FUNCTION_BLOCK LC_TOUCH (* Composite Function Block Type *)
  (* Standard: 61499-2 *)
  (* Version 0.0, 2012-01-30, 4DIAC-IDE, 4DIAC-Consortium *)
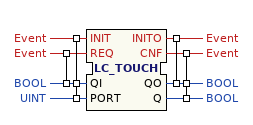
  EVENT_INPUT
    INIT WITH QI, PORT; (* Initialization Request *)
    REQ WITH QI; (* Normal Execution Request *)
  END_EVENT
  EVENT_OUTPUT
    INITO WITH QO; (* Initialization Confirm *)
    CNF WITH QO, Q; (* Execution Confirmation *)
  END_EVENT
  VAR_INPUT
    QI : BOOL; (* Input event qualifier *)
    PORT : UINT; (* Port # *)
  END_VAR
  VAR_OUTPUT
    QO : BOOL; (* Output event qualifier *)
    Q : BOOL; (* True if pressed *)
  END_VAR
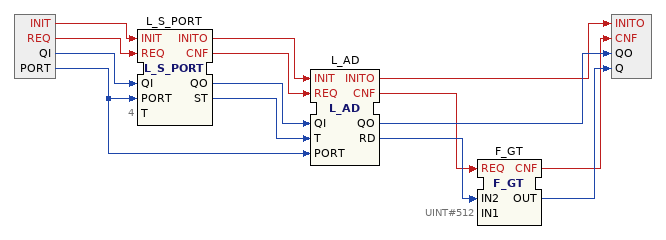
  FBS
    L_AD : L_AD;
    L_S_PORT : L_S_PORT(T := 4);
    F_GT : F_GT(IN1 := UINT#512);
  END_FBS
  EVENT_CONNECTIONS
    INIT TO L_S_PORT.INIT;
    L_S_PORT.INITO TO L_AD.INIT;
    L_AD.INITO TO INITO;
    REQ TO L_S_PORT.REQ;
    L_S_PORT.CNF TO L_AD.REQ;
    L_AD.CNF TO F_GT.REQ;
    F_GT.CNF TO CNF;
  END_CONNECTIONS
  DATA_CONNECTIONS
    L_AD.QO TO QO;
    L_S_PORT.QO TO L_AD.QI;
    L_S_PORT.ST TO L_AD.T;
    QI TO L_S_PORT.QI;
    PORT TO L_S_PORT.PORT;
    PORT TO L_AD.PORT;
    L_AD.RD TO F_GT.IN2;
    F_GT.OUT TO Q;
  END_CONNECTIONS
END_FUNCTION_BLOCK
